// TIA Portal V15.1 export
// export: Created 2024-05-17T05:38:24.7834223Z, ExportSetting WithDefaults, DisplayName Totally Integrated Automation Portal, DisplayVersion V15.1 Update 5, DisplayName TIA Portal Openness, DisplayVersion V15.1 Update 5, DisplayName SINAMICS Startdrive Advanced, DisplayVersion V15.1, DisplayName G130, G150, S120, S150, SINAMICS MV, S210, DisplayVersion V15.1, DisplayName G110M, G120, G120C, G120D, G120P, DisplayVersion V15.1, DisplayName STEP 7 Professional, DisplayVersion V15.1 Update 5, DisplayName STEP 7 Safety, DisplayVersion V15.1, DisplayName WinCC Professional, DisplayVersion V15.1 Update 5, DisplayName SIMATIC Visualization Architect, DisplayVersion V15.1
FUNCTION_BLOCK "LUps-Puls"   // FB1314, FBD
TITLE = LUps-M / LUps-M 2012-05-11 / LUps-Puls 2020-07-17
{ S7_Optimized_Access := 'FALSE' }
AUTHOR : VCC_JS
FAMILY : Actuator
NAME : LUps
VERSION : 0.2
// ================================================================================
// This module handles alarms from the UPS of type Murr electronic.
// When the conditions to generate the alarm disappear, a boolean output is 
// available to inform the upper level that the alarm can be reset.
// ================================================================================
// stored: AutoNumber false, IsIECCheckEnabled false, SetENOAutomatically False, UDAEnableTagReadback false
   VAR_INPUT
      I_Active { ExternalAccessible := 'False'; ExternalVisible := 'False'; ExternalWritable := 'False'} : Bool;   // Input signal of UPS Active-Signal / Input signal of UPS OK-signal
      I_Ready { ExternalAccessible := 'False'; ExternalVisible := 'False'; ExternalWritable := 'False'} : Bool;   // Input signal UPS Ready-Signal / Input signal supply voltage OK
      I_EnableAlarm { ExternalAccessible := 'False'; ExternalVisible := 'False'; ExternalWritable := 'False'} : Bool := TRUE;   // Enable alarm from upper level (0=disable/1=enable)
      I_AlarmResetPB { ExternalAccessible := 'False'; ExternalVisible := 'False'; ExternalWritable := 'False'} : Bool;   // Alarm reset pushbutton is activated
   END_VAR
   VAR_OUTPUT
      O_Active { ExternalAccessible := 'False'; ExternalVisible := 'False'; ExternalWritable := 'False'} : Bool;   // UPS Active / UPS ok
      O_AlarmA { ExternalAccessible := 'False'; ExternalVisible := 'False'; ExternalWritable := 'False'} : Bool;   // Summation Alarm A.
      O_AlarmB { ExternalAccessible := 'False'; ExternalVisible := 'False'; ExternalWritable := 'False'} : Bool;   // Summation Alarm B.
      O_AlarmC { ExternalAccessible := 'False'; ExternalVisible := 'False'; ExternalWritable := 'False'} : Bool;   // Summation Alarm C.
      O_AlarmD { ExternalAccessible := 'False'; ExternalVisible := 'False'; ExternalWritable := 'False'} : Bool;   // Summation Alarm D.
      O_AlarmABCondition { ExternalAccessible := 'False'; ExternalVisible := 'False'; ExternalWritable := 'False'} : Bool;   // Alarm AB Condition
      H_IAnim { ExternalAccessible := 'False'; ExternalVisible := 'False'; ExternalWritable := 'False'} : DWord;   // Icon animation
      H_AlarmWord { ExternalAccessible := 'False'; ExternalVisible := 'False'; ExternalWritable := 'False'} : DWord;   // Alarm Word
   END_VAR
   VAR DB_SPECIFIC
      AA_Active { ExternalAccessible := 'False'; ExternalVisible := 'False'; ExternalWritable := 'False'} : Bool;   // UPS Capaciter discharged / UPS Fault / 0000: UPS Fault
      AD_Ready { ExternalAccessible := 'False'; ExternalVisible := 'False'; ExternalWritable := 'False'} : Bool;   // UPS Ready-Signal / Supply voltage not Ok / 0000: Supply voltage not Ok
      H_Out : Struct   // HMI
         Anim : Word;   // HMI Animation of the object
         DBnr : Int;   // HMI Animation DB number
      END_STRUCT;
      UPSActiveAlarmCond { ExternalAccessible := 'False'; ExternalVisible := 'False'; ExternalWritable := 'False'} : Bool;   // Active condition to set the UPS alarm / Input condition to set the UPS alarm
      AlarmA { ExternalAccessible := 'False'; ExternalVisible := 'False'; ExternalWritable := 'False'} : Bool;   // Summation Alarm A
      AlarmB { ExternalAccessible := 'False'; ExternalVisible := 'False'; ExternalWritable := 'False'} : Bool;   // Summation Alarm B
      AlarmC { ExternalAccessible := 'False'; ExternalVisible := 'False'; ExternalWritable := 'False'} : Bool;   // Summation Alarm C
      AlarmD { ExternalAccessible := 'False'; ExternalVisible := 'False'; ExternalWritable := 'False'} : Bool;   // Summation Alarm D
      DBnr { ExternalAccessible := 'False'; ExternalVisible := 'False'; ExternalWritable := 'False'} : Int;   // DB number
   END_VAR
BEGIN

NETWORK
TITLE = **** 1 - Inputs **** DB number
// DB number
      L     DINO;
      T     #DBnr;

REGION Network 2: **** 1 - Inputs **** The UPS alarm is active / **** 1 - Inputs **** / **** 2.2 - Alarms - Alarms Generation **** UPS Not Active alarm condition
   // The UPS alarm is active / UPS Active alarm condition (Capacitors are  being discharged)
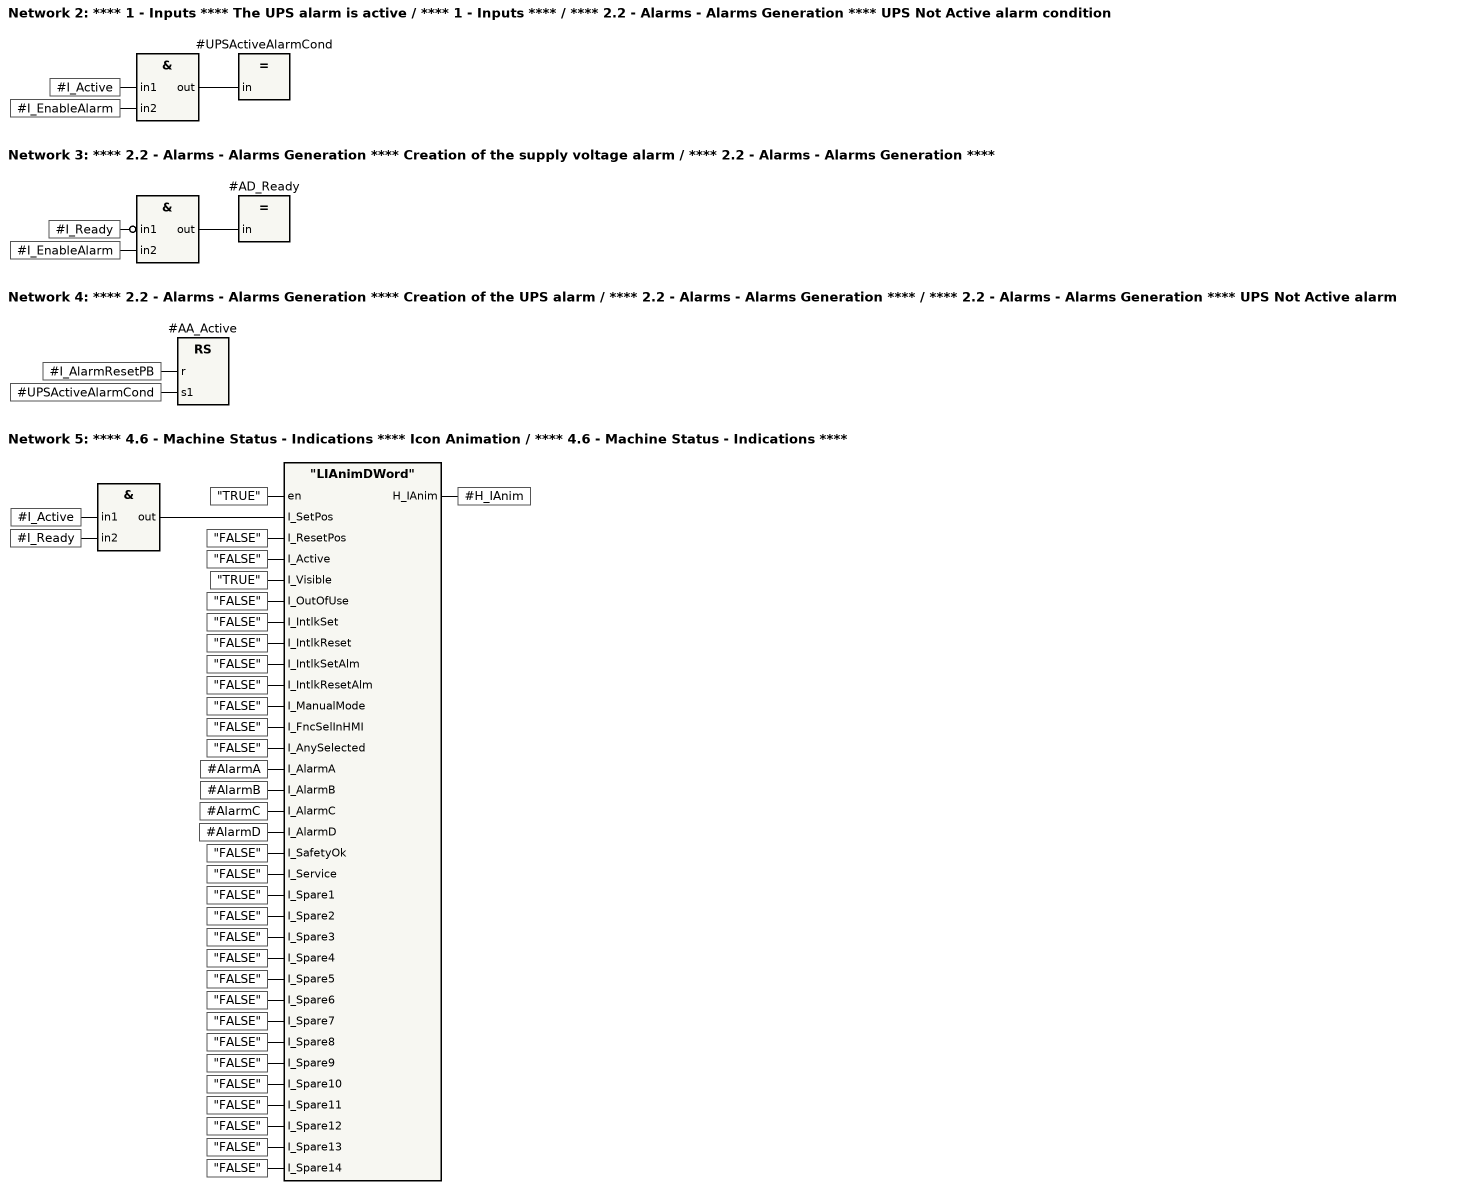
   #UPSActiveAlarmCond := #I_Active AND #I_EnableAlarm;
END_REGION

REGION Network 3: **** 2.2 - Alarms - Alarms Generation **** Creation of the supply voltage alarm / **** 2.2 - Alarms - Alarms Generation ****
   // Creation of the supply voltage alarm
   #AD_Ready := NOT #I_Ready AND #I_EnableAlarm;
END_REGION

REGION Network 4: **** 2.2 - Alarms - Alarms Generation **** Creation of the UPS alarm / **** 2.2 - Alarms - Alarms Generation **** / **** 2.2 - Alarms - Alarms Generation **** UPS Not Active alarm
   // Creation of the UPS alarm
   IF #I_AlarmResetPB THEN
       #AA_Active := FALSE;   // RS flip-flop
   END_IF;
   IF #UPSActiveAlarmCond THEN #AA_Active := TRUE; END_IF;
END_REGION

REGION Network 5: **** 4.6 - Machine Status - Indications **** Icon Animation / **** 4.6 - Machine Status - Indications ****
   // Icon Animation
   IF "TRUE" THEN
       "LIAnimDWord"(I_SetPos := #I_Active AND #I_Ready,
                     I_ResetPos := "FALSE",
                     I_Active := "FALSE",
                     I_Visible := "TRUE",
                     I_OutOfUse := "FALSE",
                     I_IntlkSet := "FALSE",
                     I_IntlkReset := "FALSE",
                     I_IntlkSetAlm := "FALSE",
                     I_IntlkResetAlm := "FALSE",
                     I_ManualMode := "FALSE",
                     I_FncSelInHMI := "FALSE",
                     I_AnySelected := "FALSE",
                     I_AlarmA := #AlarmA,
                     I_AlarmB := #AlarmB,
                     I_AlarmC := #AlarmC,
                     I_AlarmD := #AlarmD,
                     I_SafetyOk := "FALSE",
                     I_Service := "FALSE",
                     I_Spare1 := "FALSE",
                     I_Spare2 := "FALSE",
                     I_Spare3 := "FALSE",
                     I_Spare4 := "FALSE",
                     I_Spare5 := "FALSE",
                     I_Spare6 := "FALSE",
                     I_Spare7 := "FALSE",
                     I_Spare8 := "FALSE",
                     I_Spare9 := "FALSE",
                     I_Spare10 := "FALSE",
                     I_Spare11 := "FALSE",
                     I_Spare12 := "FALSE",
                     I_Spare13 := "FALSE",
                     I_Spare14 := "FALSE",
                     H_IAnim => #H_IAnim);
   END_IF;
END_REGION

REGION Network 6: **** 4.6 - Machine Status - Indications **** Animation / **** 4.6 - Machine Status - Indications ****
   // Animation
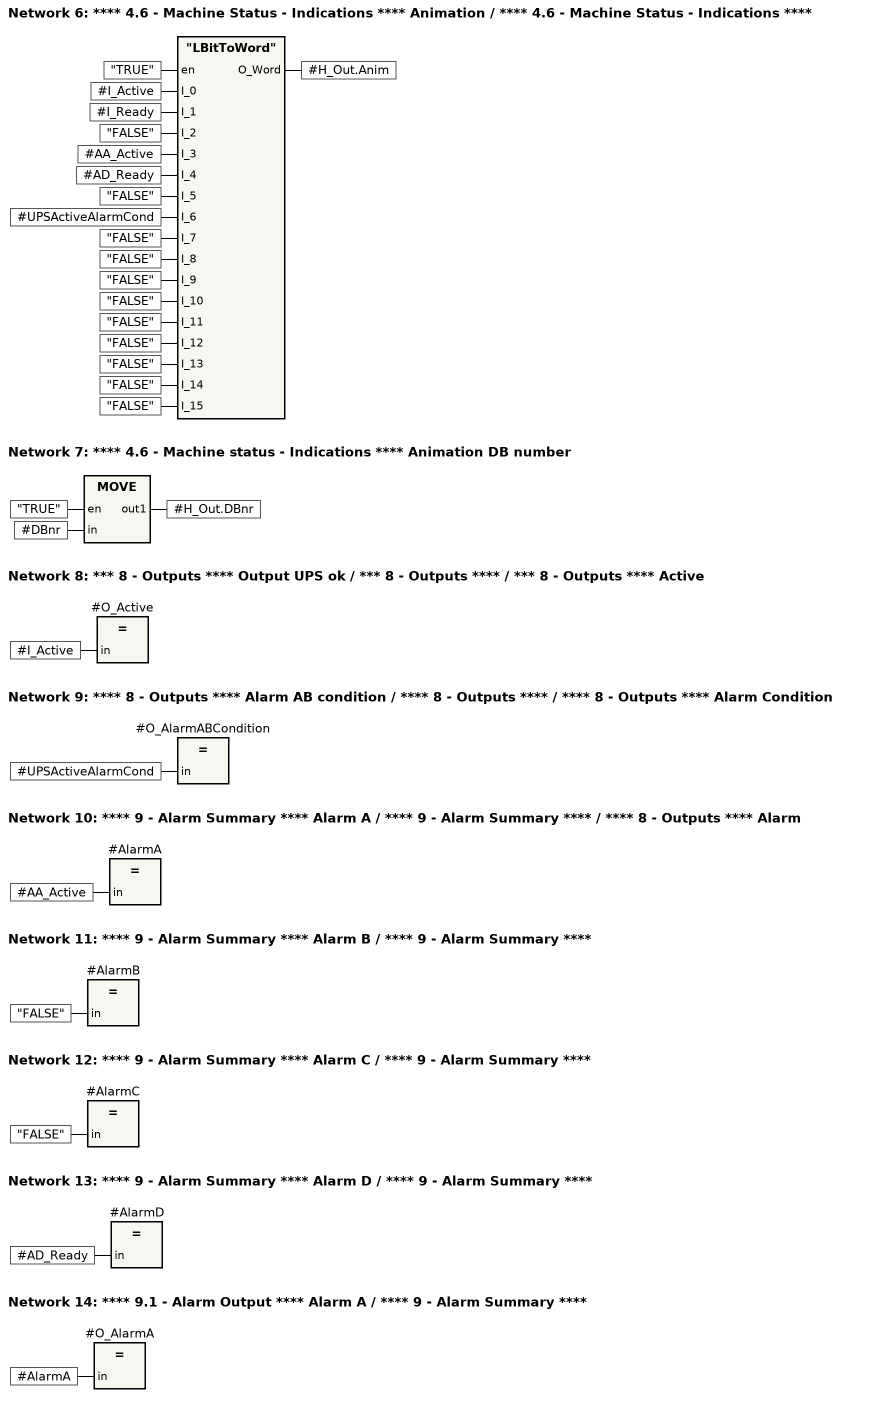
   IF "TRUE" THEN
       "LBitToWord"(I_0 := #I_Active,
                    I_1 := #I_Ready,
                    I_2 := "FALSE",
                    I_3 := #AA_Active,
                    I_4 := #AD_Ready,
                    I_5 := "FALSE",
                    I_6 := #UPSActiveAlarmCond,
                    I_7 := "FALSE",
                    I_8 := "FALSE",
                    I_9 := "FALSE",
                    I_10 := "FALSE",
                    I_11 := "FALSE",
                    I_12 := "FALSE",
                    I_13 := "FALSE",
                    I_14 := "FALSE",
                    I_15 := "FALSE",
                    O_Word => #H_Out.Anim);
   END_IF;
END_REGION

REGION Network 7: **** 4.6 - Machine status - Indications **** Animation DB number
   // Animation DB number
   IF "TRUE" THEN #H_Out.DBnr := #DBnr; END_IF;
END_REGION

REGION Network 8: *** 8 - Outputs **** Output UPS ok / *** 8 - Outputs **** / *** 8 - Outputs **** Active
   // Output UPS ok
   #O_Active := #I_Active;
END_REGION

REGION Network 9: **** 8 - Outputs **** Alarm AB condition / **** 8 - Outputs **** / **** 8 - Outputs **** Alarm Condition
   // Alarm AB Condition
   #O_AlarmABCondition := #UPSActiveAlarmCond;
END_REGION

REGION Network 10: **** 9 - Alarm Summary **** Alarm A / **** 9 - Alarm Summary **** / **** 8 - Outputs **** Alarm
   // Summary of alarms A / Alarm
   #AlarmA := #AA_Active;
END_REGION

REGION Network 11: **** 9 - Alarm Summary **** Alarm B / **** 9 - Alarm Summary ****
   // Summary of alarms B
   #AlarmB := "FALSE";
END_REGION

REGION Network 12: **** 9 - Alarm Summary **** Alarm C / **** 9 - Alarm Summary ****
   // Summary of alarms C
   #AlarmC := "FALSE";
END_REGION

REGION Network 13: **** 9 - Alarm Summary **** Alarm D / **** 9 - Alarm Summary ****
   // Summary of alarms D
   #AlarmD := #AD_Ready;
END_REGION

REGION Network 14: **** 9.1 - Alarm Output **** Alarm A / **** 9 - Alarm Summary ****
   // Output of alarms A
   #O_AlarmA := #AlarmA;
END_REGION

REGION Network 15: **** 9.1 - Alarm Output **** Alarm B / **** 9 - Alarm Summary ****
   // Output of alarms B
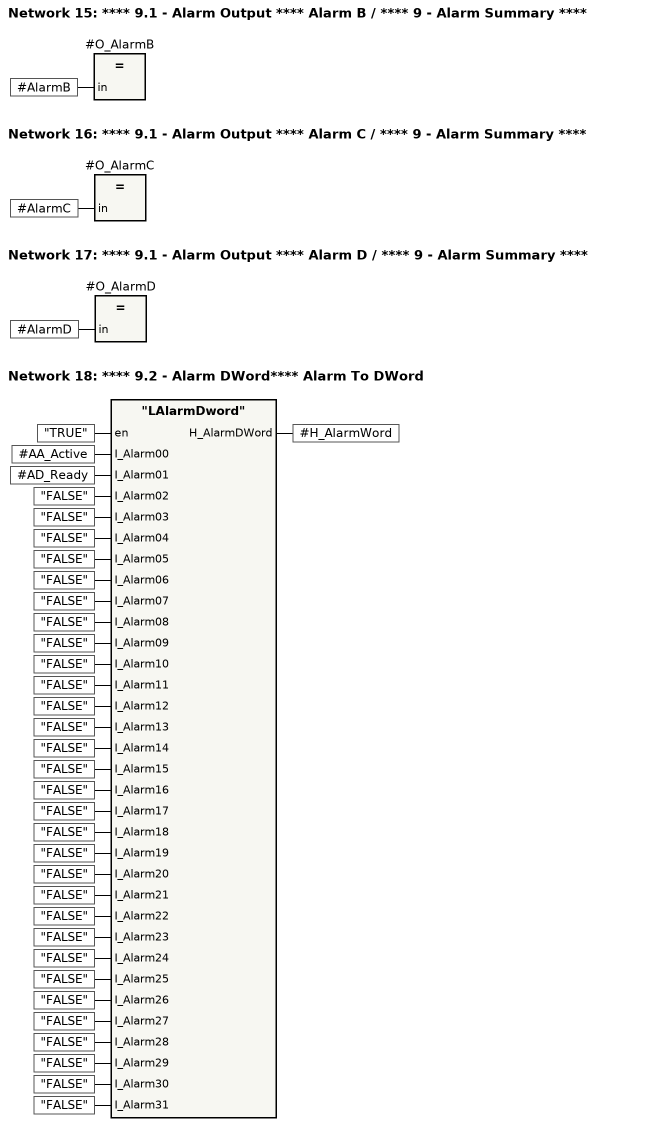
   #O_AlarmB := #AlarmB;
END_REGION

REGION Network 16: **** 9.1 - Alarm Output **** Alarm C / **** 9 - Alarm Summary ****
   // Output of alarms C
   #O_AlarmC := #AlarmC;
END_REGION

REGION Network 17: **** 9.1 - Alarm Output **** Alarm D / **** 9 - Alarm Summary ****
   // Output of alarms D
   #O_AlarmD := #AlarmD;
END_REGION

REGION Network 18: **** 9.2 - Alarm DWord**** Alarm To DWord
   // Alarm Word
   IF "TRUE" THEN
       "LAlarmDword"(I_Alarm00 := #AA_Active,
                     I_Alarm01 := #AD_Ready,
                     I_Alarm02 := "FALSE",
                     I_Alarm03 := "FALSE",
                     I_Alarm04 := "FALSE",
                     I_Alarm05 := "FALSE",
                     I_Alarm06 := "FALSE",
                     I_Alarm07 := "FALSE",
                     I_Alarm08 := "FALSE",
                     I_Alarm09 := "FALSE",
                     I_Alarm10 := "FALSE",
                     I_Alarm11 := "FALSE",
                     I_Alarm12 := "FALSE",
                     I_Alarm13 := "FALSE",
                     I_Alarm14 := "FALSE",
                     I_Alarm15 := "FALSE",
                     I_Alarm16 := "FALSE",
                     I_Alarm17 := "FALSE",
                     I_Alarm18 := "FALSE",
                     I_Alarm19 := "FALSE",
                     I_Alarm20 := "FALSE",
                     I_Alarm21 := "FALSE",
                     I_Alarm22 := "FALSE",
                     I_Alarm23 := "FALSE",
                     I_Alarm24 := "FALSE",
                     I_Alarm25 := "FALSE",
                     I_Alarm26 := "FALSE",
                     I_Alarm27 := "FALSE",
                     I_Alarm28 := "FALSE",
                     I_Alarm29 := "FALSE",
                     I_Alarm30 := "FALSE",
                     I_Alarm31 := "FALSE",
                     H_AlarmDWord => #H_AlarmWord);
   END_IF;
END_REGION
END_FUNCTION_BLOCK
